{attribute 'qualified_only'}
VAR_GLOBAL CONSTANT
	iMaxArray : INT := 5;
END_VAR

(* stored: Version 1.1.0.1, ProductVersion 3.1.4024.12
   GVL Param: Id {3b8285a4-a667-47fe-aad6-a7680751710e}, ParameterList True *)
